FUNCTION TryConvert_DWORD_TO_DT : BOOL
VAR_INPUT
	in : DWORD;
	out : REFERENCE TO DT;
END_VAR

out := DWORD_TO_DT(in);
TryConvert_DWORD_TO_DT := TRUE;

END_FUNCTION

(* stored: Version 1.1.0.1, ProductVersion 3.1.4024.12
   POU TryConvert_DWORD_TO_DT: Id {2a291cec-06e2-4d9a-a14f-7b4a09752732}, SpecialFunc None *)
